# EPICS substitutions: BLDApp/Db/eOrbitsFcomSim.substitutions
#
# Sample substitutions file to create and send dummy fcom blob groups
#
# Data values alternate between sin and cos calc records
# advancing 1 degree per upate at 120hz
#

file fcomBlobAo.template
{
	pattern
	{	P,			SIM,	INDEX,	GROUP,	BLOB				}
	{	"$(BLOB)",	"_SIM",		0,		0,	BPMS:LTU1:910:X		}
	{	"$(BLOB)",	"_SIM",		1,		0,	BPMS:LTU1:910:Y		}
	{	"$(BLOB)",	"_SIM",		2,		0,	BPMS:LTU1:910:T		}

	{	"$(BLOB)",	"_SIM",		0,		0,	BPMS:LTU1:960:X		}
	{	"$(BLOB)",	"_SIM",		1,		0,	BPMS:LTU1:960:Y		}
	{	"$(BLOB)",	"_SIM",		2,		0,	BPMS:LTU1:960:T		}

	{	"$(BLOB)",	"_SIM",		0,		0,	BPMS:UND1:100:X		}
	{	"$(BLOB)",	"_SIM",		1,		0,	BPMS:UND1:100:Y		}
	{	"$(BLOB)",	"_SIM",		2,		0,	BPMS:UND1:100:T		}

	{	"$(BLOB)",	"_SIM",		0,		0,	BPMS:UND1:190:X		}
	{	"$(BLOB)",	"_SIM",		1,		0,	BPMS:UND1:190:Y		}
	{	"$(BLOB)",	"_SIM",		2,		0,	BPMS:UND1:190:T		}

	{	"$(BLOB)",	"_SIM",		0,		0,	BPMS:UND1:290:X		}
	{	"$(BLOB)",	"_SIM",		1,		0,	BPMS:UND1:290:Y		}
	{	"$(BLOB)",	"_SIM",		2,		0,	BPMS:UND1:290:T		}

	{	"$(BLOB)",	"_SIM",		0,		0,	BPMS:UND1:390:X		}
	{	"$(BLOB)",	"_SIM",		1,		0,	BPMS:UND1:390:Y		}
	{	"$(BLOB)",	"_SIM",		2,		0,	BPMS:UND1:390:T		}

	{	"$(BLOB)",	"_SIM",		0,		1,	BPMS:UND1:490:X		}
	{	"$(BLOB)",	"_SIM",		1,		1,	BPMS:UND1:490:Y		}
	{	"$(BLOB)",	"_SIM",		2,		1,	BPMS:UND1:490:T		}

	{	"$(BLOB)",	"_SIM",		0,		1,	BPMS:UND1:590:X		}
	{	"$(BLOB)",	"_SIM",		1,		1,	BPMS:UND1:590:Y		}
	{	"$(BLOB)",	"_SIM",		2,		1,	BPMS:UND1:590:T		}

	{	"$(BLOB)",	"_SIM",		0,		1,	BPMS:UND1:690:X		}
	{	"$(BLOB)",	"_SIM",		1,		1,	BPMS:UND1:690:Y		}
	{	"$(BLOB)",	"_SIM",		2,		1,	BPMS:UND1:690:T		}

	{	"$(BLOB)",	"_SIM",		0,		1,	BPMS:UND1:790:X		}
	{	"$(BLOB)",	"_SIM",		1,		1,	BPMS:UND1:790:Y		}
	{	"$(BLOB)",	"_SIM",		2,		1,	BPMS:UND1:790:T		}

	{	"$(BLOB)",	"_SIM",		0,		1,	BPMS:UND1:890:X		}
	{	"$(BLOB)",	"_SIM",		1,		1,	BPMS:UND1:890:Y		}
	{	"$(BLOB)",	"_SIM",		2,		1,	BPMS:UND1:890:T		}

	{	"$(BLOB)",	"_SIM",		0,		1,	BPMS:UND1:990:X		}
	{	"$(BLOB)",	"_SIM",		1,		1,	BPMS:UND1:990:Y		}
	{	"$(BLOB)",	"_SIM",		2,		1,	BPMS:UND1:990:T		}

}

#file fcomBlobAdd.template
#{
#	pattern
#	{	P,			R,		GROUP,	BLOB				}
#	{	"$(BLOB)",	"_ADD",		0,	BPMS:LTU1:910:ALL	}
#	{	"$(BLOB)",	"_ADD",		0,	BPMS:LTU1:960:ALL	}
#	{	"$(BLOB)",	"_ADD",		0,	BPMS:UND1:100:ALL	}
#	{	"$(BLOB)",	"_ADD",		0,	BPMS:UND1:190:ALL	}
#	{	"$(BLOB)",	"_ADD",		0,	BPMS:UND1:290:ALL	}
#	{	"$(BLOB)",	"_ADD",		0,	BPMS:UND1:390:ALL	}
#
#	{	"$(BLOB)",	"_ADD",		1,	BPMS:UND1:490:ALL	}
#	{	"$(BLOB)",	"_ADD",		1,	BPMS:UND1:590:ALL	}
#	{	"$(BLOB)",	"_ADD",		1,	BPMS:UND1:690:ALL	}
#	{	"$(BLOB)",	"_ADD",		1,	BPMS:UND1:790:ALL	}
#	{	"$(BLOB)",	"_ADD",		1,	BPMS:UND1:890:ALL	}
#	{	"$(BLOB)",	"_ADD",		1,	BPMS:UND1:990:ALL	}
#}

# Each fcomBlobBPMS_SIM.db can be used to assign
# alternating SIN and COS values to each value in the blob,
# for up to 10 values per blob
#
# Blob macros here should truncate the value name and end w/ a colon
# i.e. BPMS:LTU0:910: instead of BPMS:LTU0:910:X
#
# The first blob in each group should define these macros
# to initiate processing of each blob where EC must be
# defined later via a dbLoadRecord macro.
#		SCAN	= "Event",	EC = "\$(EC)"
#
# Each blob in a group should specify the next
# blob in the group via a NEXT macro to force them to
# be processed sequentially.
# Leave NEXT undefined for the last blob in the group
# and it will default an FLNK to the group's send record
file fcomBlobBPMS_SIM.db
{
# group 0, six blobs
	{
		GROUP	= "0",
		SCAN	= "Event",	EC = "\$(EC)"
		BLOB	= "BPMS:LTU1:910:",
		L1		= "$(BLOB)X_SIM PP",
		L2		= "$(BLOB)Y_SIM PP",
		L3		= "$(BLOB)T_SIM PP",
		NEXT	= "BPMS:LTU1:960:SIM_SEQ"
	}
	{
		GROUP	= "0",
		BLOB	= "BPMS:LTU1:960:",
		L1		= "$(BLOB)X_SIM PP",
		L2		= "$(BLOB)Y_SIM PP",
		L3		= "$(BLOB)T_SIM PP",
		NEXT	= "BPMS:UND1:100:SIM_SEQ"
	}
	{
		GROUP	= "0",
		BLOB	= "BPMS:UND1:100:",
		L1		= "$(BLOB)X_SIM PP",
		L2		= "$(BLOB)Y_SIM PP",
		L3		= "$(BLOB)T_SIM PP",
		NEXT	= "BPMS:UND1:190:SIM_SEQ"
	}
	{
		GROUP	= "0",
		BLOB	= "BPMS:UND1:190:",
		L1		= "$(BLOB)X_SIM PP",
		L2		= "$(BLOB)Y_SIM PP",
		L3		= "$(BLOB)T_SIM PP",
		NEXT	= "BPMS:UND1:290:SIM_SEQ"
	}
	{
		GROUP	= "0",
		BLOB	= "BPMS:UND1:290:",
		L1		= "$(BLOB)X_SIM PP",
		L2		= "$(BLOB)Y_SIM PP",
		L3		= "$(BLOB)T_SIM PP",
		NEXT	= "BPMS:UND1:390:SIM_SEQ"
	}
	{
		GROUP	= "0",
		BLOB	= "BPMS:UND1:390:",
		L1		= "$(BLOB)X_SIM PP",
		L2		= "$(BLOB)Y_SIM PP",
		L3		= "$(BLOB)T_SIM PP",
		NEXT	= "BPMS:UND1:390:ALL_SEND",
	}

# Second group, six blobs
	{
		SCAN	= "Event",	EC = "\$(EC)"
		GROUP	= "1",
		BLOB	= "BPMS:UND1:490:",
		L1		= "$(BLOB)X_SIM PP",
		L2		= "$(BLOB)Y_SIM PP",
		L3		= "$(BLOB)T_SIM PP",
		NEXT	= "BPMS:UND1:590:SIM_SEQ"
	}
	{
		GROUP	= "1",
		BLOB	= "BPMS:UND1:590:",
		L1		= "$(BLOB)X_SIM PP",
		L2		= "$(BLOB)Y_SIM PP",
		L3		= "$(BLOB)T_SIM PP",
		NEXT	= "BPMS:UND1:690:SIM_SEQ"
	}
	{
		GROUP	= "1",
		BLOB	= "BPMS:UND1:690:",
		L1		= "$(BLOB)X_SIM PP",
		L2		= "$(BLOB)Y_SIM PP",
		L3		= "$(BLOB)T_SIM PP",
		NEXT	= "BPMS:UND1:790:SIM_SEQ"
	}
	{
		GROUP	= "1",
		BLOB	= "BPMS:UND1:790:",
		L1		= "$(BLOB)X_SIM PP",
		L2		= "$(BLOB)Y_SIM PP",
		L3		= "$(BLOB)T_SIM PP",
		NEXT	= "BPMS:UND1:890:SIM_SEQ"
	}
	{
		GROUP	= "1",
		BLOB	= "BPMS:UND1:890:",
		L1		= "$(BLOB)X_SIM PP",
		L2		= "$(BLOB)Y_SIM PP",
		L3		= "$(BLOB)T_SIM PP",
		NEXT	= "BPMS:UND1:990:SIM_SEQ"
	}
	{
		GROUP	= "1",
		BLOB	= "BPMS:UND1:990:",
		L1		= "$(BLOB)X_SIM PP",
		L2		= "$(BLOB)Y_SIM PP",
		L3		= "$(BLOB)T_SIM PP",
		NEXT	= "BPMS:UND1:990:ALL_SEND",
	}
}

# Each group needs a SEND record
# LAST should match the truncated BLOB macro
# from above for the last blob in the group
file fcomGroupSend.template
{
	{
		GROUP	= "0",
		LAST	= "BPMS:UND1:390:",
	}
	{
		GROUP	= "1",
		LAST	= "BPMS:UND1:990:",
	}
}
